FUNCTION_BLOCK INIT_ARR_0028_BYTE (* FB to make an Array (generic FB) *)
  (* Standard: 61499-2; Description: Copyright (c) 2026 Andreas Demmler Fahrzeugbau This program and the accompanying materials are made available under the terms of the Eclipse Public License 2.0 which is available at https://www.eclipse.org/legal/epl-2.0/ SPDX-License-Identifier: EPL-2.0 Can have a Initial Value e.g. [16#01, 16#00, 16#00, 16#00, 16#00, 16#AA, 16#00, 16#00, ...] on the Input of the in/out *)
  (* Version 1.0, 2026-01-22, Franz Höpfinger, Andreas Demmler Fahrzeugbau *)
  PACKAGE eclipse4diac::convert::generate;
  {SET_ATTRIBUTE(eclipse4diac::core::GenericClassName, 'GEN_INIT_ARR')}
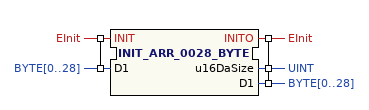
  EVENT_INPUT
    INIT : EInit WITH D1; (* Service Initialization *)
  END_EVENT
  EVENT_OUTPUT
    INITO : EInit WITH u16DaSize, D1; (* Initialization Confirm *)
  END_EVENT
  VAR_OUTPUT
    u16DaSize : UINT; (* Data length in Array Elements *)
  END_VAR
  VAR_IN_OUT
    D1 : ARRAY [0..28] OF BYTE; (* Array in/out *)
  END_VAR
END_FUNCTION_BLOCK
